TYPE InputBase_8311D824 :
STRUCT
END_STRUCT
END_TYPE

(* stored: Version 1.2.0.0, ProductVersion 3.1.4024.9
   DUT InputBase_8311D824: Id {4e289d91-0e87-4467-a729-6e50ad634c2e} *)
